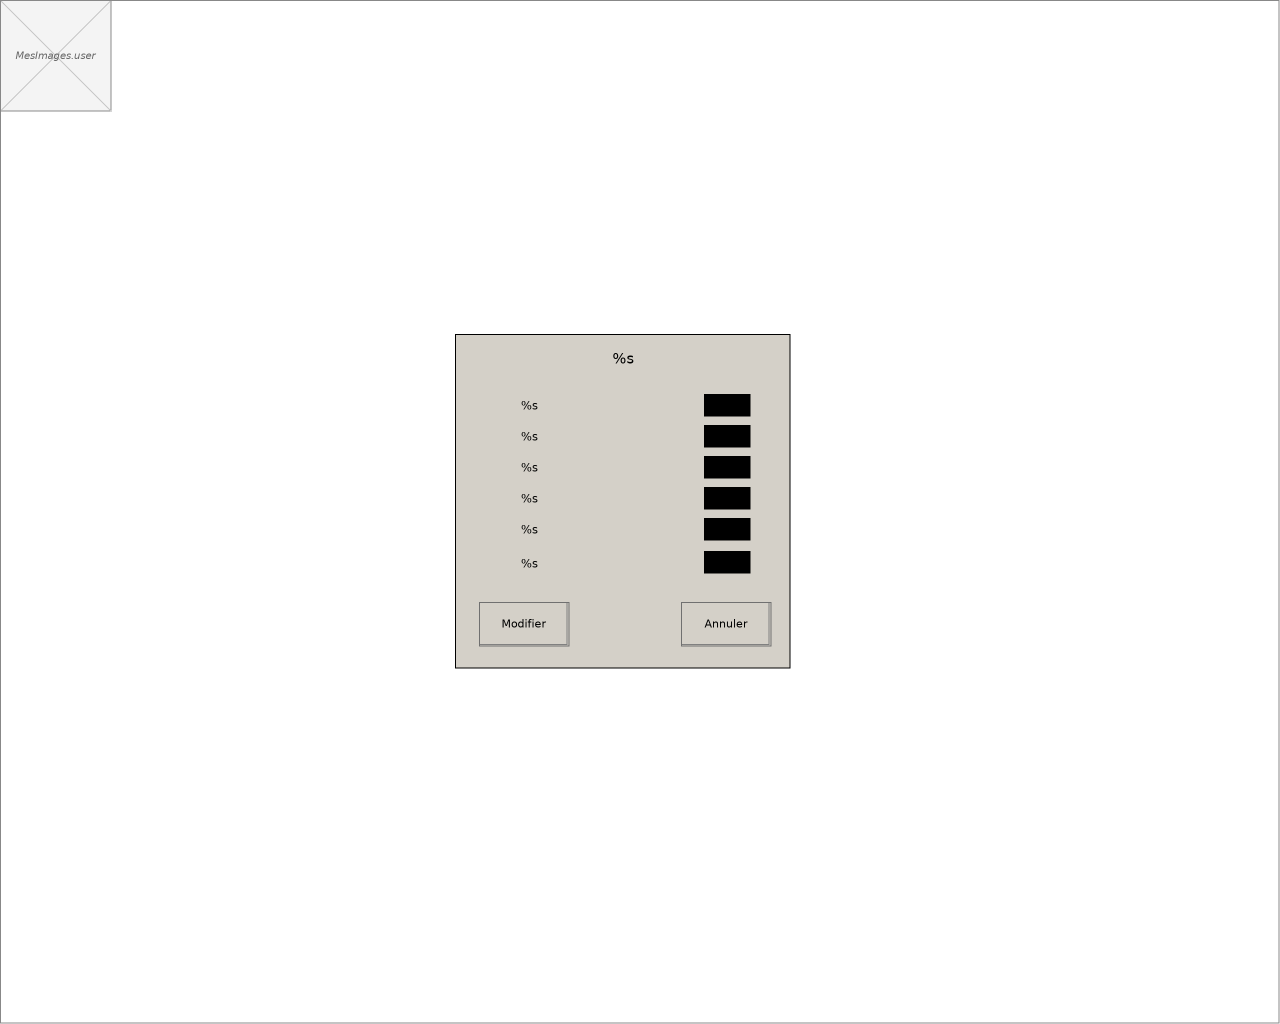
VISUALIZATION UTIL_DEFAUT  // 1280x1024
    Image (0,0 111x111), image: MesImages.user
    RoundedRectangle (455,334 335x334)
    Rectangle (460,344 327x29), "%s", text list: 'TextList_Util_Defaut', text index: 1
    Rectangle (518,422 112x29), "%s", text list: 'TextList_Util_Group', text index: 4
    Rectangle (518,453 112x29), "%s", text list: 'TextList_Util_Group', text index: 5
    Rectangle (518,391 112x29), "%s", text list: 'TextList_Util_Group', text index: 3
    Rectangle (518,484 112x29), "%s", text list: 'TextList_Util_Group', text index: 6
    Rectangle (518,515 112x29), "%s", text list: 'TextList_Util_Group', text index: 7
    Rectangle (518,549 122x29), "%s", text list: 'TextList_Util_Group', text index: 8
    Rectangle (704,394 46x22), "Oui", colour toggle: Global_Variables.PRG_USER.GROUP_TEMP.PROGRAMMATION
        toggle Global_Variables.PRG_USER.GROUP_TEMP.PROGRAMMATION
    Rectangle (704,425 46x22), "Oui", colour toggle: Global_Variables.PRG_USER.GROUP_TEMP.MAINTENANCE
        toggle Global_Variables.PRG_USER.GROUP_TEMP.MAINTENANCE
    Rectangle (704,456 46x22), "Oui", colour toggle: Global_Variables.PRG_USER.GROUP_TEMP.SUPERVISEUR
        toggle Global_Variables.PRG_USER.GROUP_TEMP.SUPERVISEUR
    Rectangle (704,487 46x22), "Oui", colour toggle: Global_Variables.PRG_USER.GROUP_TEMP.PRODUCTION
        toggle Global_Variables.PRG_USER.GROUP_TEMP.PRODUCTION
    Rectangle (704,518 46x22), "Oui", colour toggle: Global_Variables.PRG_USER.GROUP_TEMP.CONF_MACHINE
        toggle Global_Variables.PRG_USER.GROUP_TEMP.CONF_MACHINE
    Rectangle (704,551 46x22), "Oui", colour toggle: Global_Variables.PRG_USER.GROUP_TEMP.FONCTION_SA
        toggle Global_Variables.PRG_USER.GROUP_TEMP.FONCTION_SA
    Button (479,602 90x44), "Modifier"
        toggle PRG_USER.DD_mod_def2
        OnMouseClick: change screen: UTIL_MENU
    Button (681,602 90x44), "Annuler"
        OnMouseClick: change screen: UTIL_MENU
END_VISUALIZATION

(* stored: Version 1.1.0.1, ProductVersion 3.1.4024.10
   Visu UTIL_DEFAUT: Id {1d7c8725-6ec1-44d0-bffb-147ee70531a7} *)
